RoboDK station: Program without holes and paths.rdk

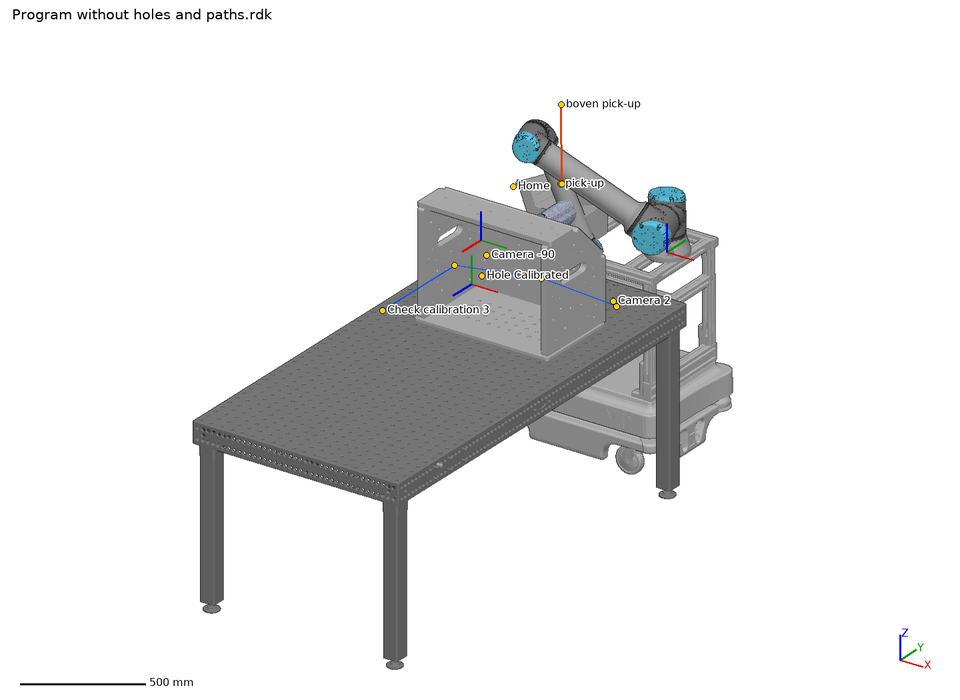
[picture v0: the station drawn from its stored meshes, robots at their saved joint values, targets as dots, program paths as lines]
Station Program without holes and paths (saved by RoboDK 5.7.0). Poses are relative to the parent item; angles as X-Y-Z fixed-axis rotations.
Station parameters (name, value as stored): 0.4, 1, 1, CollisionFreePlanner, UR10e, CollisionFreePlanner-Rob UR10e, Simplify-Mesh-Settings
  - object Lastafel at (0, 0, 0) mm, size 1021.8 x 2000 x 842 mm
  - object Lastafel_simplified at (0, 0, 0) mm, size 1000 x 2000 x 802.1 mm
  - frame UR10e Base at (-300, 2141.5, 91.6) mm, rotated rx 0.6 ry -0.16 rz 0 deg
    - robot UR10e: 6 axes, payload 10 kg, reach 1300 mm, repeatability 0.05 mm, weight 28.9 kg
        modified DH rows (alpha deg, a mm, theta deg, d mm): 0, 0, 0, 180.7; 90, 0, 180, 0; 0, 612.6, 0, 0; 0, 571.335, 0, 174.15; -90, 0, 0, 119.85; 90, 0, 180, 116.55
        joint limits [-70, -140, 0, -220, -180, -280] to [85, 0, 170, 200, 180, 115]; home [30.872, -95.296, 116.362, -22.187, 121.11, 179.827]; saved at [19.93, -32.205, 143.342, -201.422, 90.448, -19.841]
      - tool Screwdriver indraaitool, TCP at (215, -0.23, 99.66) mm, rotated rx 0 ry 90 rz 0 deg, size 345 x 117.4 x 144.9 mm, geometry from 0 Screwdriver assembly.STEP
      - tool Camera, TCP at (304, 50.7, 13.6) mm, rotated rx 0 ry 90 rz 0 deg
      - tool pointer, TCP at (196, -0.23, 99.66) mm, rotated rx 0 ry 90 rz 0 deg
      - tool Screwdriver simplified, TCP at (0, 0, 220) mm, size 159.8 x 129.1 x 379.7 mm, geometry from Screwdriver simplified.stl
      - tool indraaien, TCP at (205, 0.2, 100) mm, rotated rx 0 ry 90 rz 0 deg
    - object Assembly mir + frame aangepast naar ur10e versie 2 at (-733.08, 277.19, -552.66) mm, rotated rx 90 ry 0 rz 0.45 deg, size 901.1 x 1139.6 x 580.4 mm, geometry from Assembly mir + frame aangepast naar ur10e versie 2.STEP
    - object Mir + frame simplified at (-733.08, 277.19, -552.66) mm, rotated rx 90 ry 0 rz 0.45 deg, size 925.7 x 1139.7 x 582 mm
    - target boven pick-up (joint target) at (-657.55, 210.4, 385.42) mm, rotated rx 180 ry -0.01 rz 58.34 deg; joints [-50.868, -81.351, 94.607, -13.692, -19.23, -89.565] of UR10e
    - target pick-up (joint target) at (-663.21, 209.22, 32.36) mm, rotated rx 179.99 ry 0 rz 58.33 deg; joints [-50.468, -67.472, 110.452, -43.416, -18.832, -89.554] of UR10e
    - target unclamped (joint target) at (-658.69, 209.89, 32.4) mm, rotated rx -180 ry 0 rz 58.34 deg; joints [-50.794, -47.979, 113.128, 114.877, 19.182, -270.008] of UR10e
  - frame Hoek lastafel at (-1020, 1876.5, 50) mm, rotated rx 0 ry 0 rz -90 deg
    - frame CSV Frame at (350, 200, 0) mm, rotated rx 90 ry 0 rz 90 deg
      - object Test object at (0, 0.01, 0) mm, size 650 x 517 x 400 mm, geometry from Test object.STEP
      - object Test object simplified at (0, 0.01, 0) mm, size 650.1 x 517 x 436.5 mm
      - frame Type 13 at (0, 0, 0) mm
        - target Hole Calibrated (Cartesian target) at (50, 50, 0) mm; joints [37.4, -56.56, 134.464, -78.09, 127.804, 0.412] of UR10e
    - target Camera -90 (Cartesian target) at (100, 100, 0) mm, rotated rx 180 ry 0 rz 90 deg; joints [15.382, -77.593, 120.955, -43.48, 105.947, -89.524] of UR10e
    - target Camera +90 (Cartesian target) at (100, 100, 0) mm, rotated rx -180 ry 0 rz -90 deg; joints [17.251, -55.937, 87.569, -31.877, -72.203, -90.48] of UR10e
    - target Camera Calibration (Cartesian target) at (100, 100, 0) mm, rotated rx -180 ry 0 rz 180 deg; joints [5.018, -68.171, 107.665, -44.191, 5.596, -85.486] of UR10e
    - target Camera 2 (Cartesian target) at (150, 750, 0) mm, rotated rx 180 ry 0 rz 180 deg; joints [50.749, -60.173, 157.418, 81.984, -51.264, -269.754] of UR10e
    - target Check calibration 0 (Cartesian target) at (200, 800, 10) mm, rotated rx 180 ry 0 rz 180 deg; joints [69.087, -96.044, 157.848, -62.324, 69.685, -90.102] of UR10e
    - target Check calibration 1 (Cartesian target) at (150, 400, 2) mm, rotated rx 180 ry 0 rz 180 deg; joints [4.739, -84.216, 147.782, -67.962, 5.34, -85.787] of UR10e
    - target Check calibration 2 (Cartesian target) at (250, 50, 2) mm, rotated rx 180 ry 0 rz 180 deg; joints [9.934, -58.947, 106.867, -51.902, 9.691, -86.238] of UR10e
    - target Check calibration 3 (Cartesian target) at (750, 50, 2) mm, rotated rx 180 ry 0 rz 180 deg; joints [40.424, -35.05, 60.293, -26.389, 40.152, -89.277] of UR10e
    - target Home (Cartesian target) at (200, 300, 400) mm, rotated rx 180 ry 0 rz 180 deg; joints [9.713, -85.986, 130.341, 132.467, -10.3, 92.957] of UR10e
  - program Check XY-calibration (7 instructions, listed below)
  - program helicoil pickup (9 instructions, listed below)
  - Python program retract shank (listed below)
  - Python program get_helicoil (listed below)
  - Python program Insert helicoil (listed below)
  - Python program pickup helicoil (listed below)
  - Python program Test get screwdriver data (listed below)
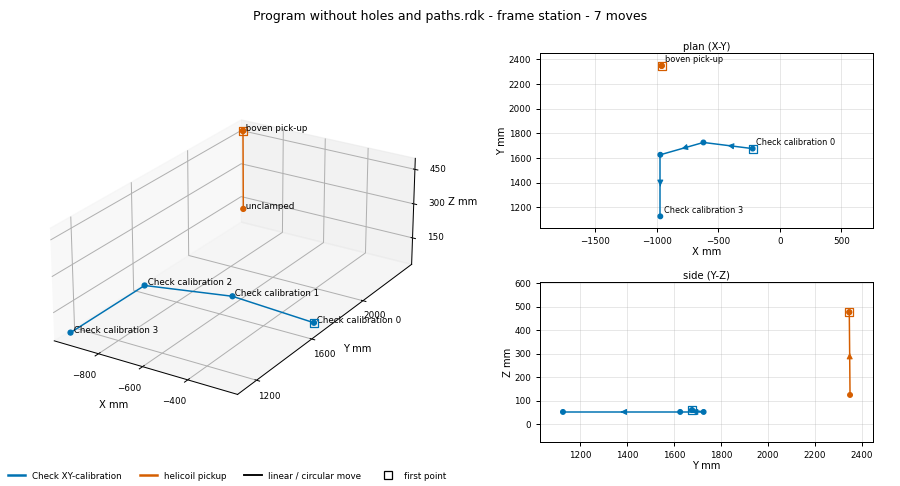
[picture p0: tool path of Program without holes and paths.rdk in frame station, 7 of 8 moves have a stored position in this frame; points joined in program order, loops and branches not executed]

--- program Check XY-calibration (robot UR10e) ---
  Set Ref.: Hoek lastafel
  Set Tool: pointer
  Set speed (200.0 mm/s)
  MoveL (Check calibration 0)
  MoveL (Check calibration 1)
  MoveL (Check calibration 2)
  MoveL (Check calibration 3)

--- program helicoil pickup (robot UR10e) ---
  Set Ref.: UR10e Base
  Set Tool: Screwdriver indraaitool
  MoveL (boven pick-up)
  Call retract shank
  MoveL (pick-up) [its target is no longer in the station]
  Call get_helicoil
  MoveL (unclamped)
  Call retract shank
  MoveL (boven pick-up)

--- Python program retract shank ---
from robodk import robolink, robomath
import time
import requests
RDK = robolink.Robolink()
robot = RDK.Item('UR10e')

# Screwdriver data
compute_box_ip = "192.168.12.15"
username = "admin"
password = "OnRobotPerron038"
tool_id = 0  # ID of the tool

#default parameters screwdriver
shaft_value = 0 #shaft position

# URL's for screwdriver commands
shank_url =  f"http://{compute_box_ip}/api/dc/sd/move_shank/{tool_id}/{shaft_value}"


#---Main Program---

#Retract shank
requests.get(shank_url, auth=(username, password))
time.sleep(1) # 1s delay
print('klaar')

--- Python program get_helicoil ---
from robodk import robolink, robomath
import time
import requests
RDK = robolink.Robolink()
robot = RDK.Item('UR10e')

DEBUG=True
if DEBUG:
    RDK.setRunMode(robolink.RUNMODE_RUN_ROBOT) #Programma wordt uitgevoerd op de robot wanneer afgespeeld vanuit de editor

#Screwdriver data
compute_box_ip = "192.168.12.15"
username = "admin"
password = "OnRobotPerron038"
tool_id = 0  # ID of the tool

#default parameters screwdriver
max_torque = .2 #max torque untill stopping screw motion via default premount behavior
screw_length = 20 #helicoil length
target_torque = 1 #target torque to stop the screw motion early via monitoring current torque and no shank motion
shank_force = 20 #shank force
shaft_value = 0

# URL's for screwdriver commands
tighten_url = f"http://{compute_box_ip}/api/dc/sd/tighten/{tool_id}/{shank_force}/{screw_length}/{max_torque}"
shank_url =  f"http://{compute_box_ip}/api/dc/sd/move_shank/{tool_id}/{shaft_value}"


#---Main Program---
print('main program')
helicoil_detect = robot.getDI(0) #output is een string: '0.000000' of '1.000000'

#get helicoil from stepfeeder
if helicoil_detect != '1.000000':
    #Move actuator
    robot.setDO(2, 1)
    robot.setDO(4, 0)
    time.sleep(4)
    #trigger feeder
    robot.setAO(0, 0.4)

#wait until helicoil is detected
helicoil_detect = robot.getDI(0)
while helicoil_detect != '1.000000':
    time.sleep(0.1)
    helicoil_detect = robot.getDI(0)

#stop feeder
robot.setAO(0, 0)

#move cylinder out
robot.setDO(2, 0)
robot.setDO(4, 1)
time.sleep(5)

#Screw on helicoil
requests.get(tighten_url, auth=(username, password))
time.sleep(3)
shaft_value=24
shank_url =  f"http://{compute_box_ip}/api/dc/sd/move_shank/{tool_id}/{shaft_value}"
requests.get(shank_url, auth=(username, password))
time.sleep(1)

#Unclamp helicoil
robot.setDO(4, 0)
robot.setDO(2, 1)
time.sleep(.1)
robot.setDO(2, 0)

--- Python program Insert helicoil ---
from robodk import robolink, robomath
import time
import requests
import tkinter as tk
from tkinter import messagebox

RDK = robolink.Robolink()
robot = RDK.Item('UR10e')

DEBUG=True
if DEBUG:
    RDK.setRunMode(robolink.RUNMODE_RUN_ROBOT) #Programma wordt uitgevoerd op de robot wanneer afgespeeld vanuit de editor

#Screwdriver data
compute_box_ip = "192.168.12.15"
username = "admin"
password = "OnRobotPerron038"
tool_id = 0  # ID of the tool

#default parameters screwdriver
shank_force = 20 #shank force
screw_length = 20 #helicoil length
max_torque = 1.5 #max torque untill stopping screw motion via default premount behavior
unscrewing_length_mm = 20
shaft_value = 0 #shank position

# URL's for screwdriver commands
tighten_url = f"http://{compute_box_ip}/api/dc/sd/tighten/{tool_id}/{shank_force}/{screw_length}/{max_torque}"
shank_url =  f"http://{compute_box_ip}/api/dc/sd/move_shank/{tool_id}/{shaft_value}"
unscrew_url = f"http://{compute_box_ip}/api/dc/sd/loosen/{tool_id}/{shank_force}/{unscrewing_length_mm}"

#---Main Program---
shaft_value = 10
shank_url =  f"http://{compute_box_ip}/api/dc/sd/move_shank/{tool_id}/{shaft_value}"
requests.get(shank_url, auth=(username, password))

root = tk.Tk()
root.withdraw()
messagebox.showinfo("Notification", "Is the tool well aligned with the hole?")
root.destroy()
time.sleep(5)


requests.get(tighten_url, auth=(username, password))
time.sleep(13)

requests.get(unscrew_url, auth=(username, password))
time.sleep(8)

shaft_value = 0
shank_url =  f"http://{compute_box_ip}/api/dc/sd/move_shank/{tool_id}/{shaft_value}"
requests.get(shank_url, auth=(username, password))
time.sleep(2)

--- Python program pickup helicoil ---
import tkinter as tk
from tkinter import messagebox

# Hide the main tkinter window
root = tk.Tk()
root.withdraw()

# Trigger the message box
messagebox.showinfo("Notification", "Is the helicoil screwed onto the tool?")

# Close the hidden window
root.destroy()

--- Python program Test get screwdriver data ---
from robodk import robolink, robomath
import time
import requests
RDK = robolink.Robolink()
robot = RDK.Item('UR10e')

DEBUG=True
if DEBUG:
    RDK.setRunMode(robolink.RUNMODE_RUN_ROBOT) #Programma wordt uitgevoerd op de robot wanneer afgespeeld vanuit de editor

#Screwdriver data
compute_box_ip = "192.168.12.15"
username = "admin"
password = "OnRobotPerron038"
tool_id = 0  # ID of the tool

#default parameters screwdriver
shank_force = 20 #shank force
screw_length = 18 #helicoil length
max_torque = 1.5 #max torque untill stopping screw motion via default premount behavior
unscrewing_length_mm = 20
shaft_value = 0 #shank position

# URL's for screwdriver commands
tighten_url = f"http://{compute_box_ip}/api/dc/sd/tighten/{tool_id}/{shank_force}/{screw_length}/{max_torque}"
shank_url =  f"http://{compute_box_ip}/api/dc/sd/move_shank/{tool_id}/{shaft_value}"
unscrew_url = f"http://{compute_box_ip}/api/dc/sd/loosen/{tool_id}/{shank_force}/{unscrewing_length_mm}"

# URL's to get screwdriver data
busy_url = f"http://{compute_box_ip}/api/dc/sd/status/{tool_id}"


#---Main Program---
response = requests.get(busy_url, auth=(username, password))
print(response)
